Fanuc KAREL source: ko00023.KL

-- PROVISIONAL review KL for V1013-1; original PC SHA256 bdae2d59f309a1ab0a29936beee89b0a31427c261c2ddde664e6fcefbd9250d4
-- Incomplete behavior may be omitted. Consult companion uncertainty JSON. Do not deploy.
PROGRAM KO00023
%NOLOCKGROUP
-- UNRESOLVED_DECL P1 type=000106
-- UNRESOLVED_DECL P2 type=000106
-- UNRESOLVED_DECL P3 type=000106
-- UNRESOLVED_DECL P4 type=000106
-- UNRESOLVED_DECL OUT type=000106
BEGIN
  -- UNRESOLVED_PC offsets 5-80; opcodes 27,27,49,7E,AD,27,49,7E,AD,27,49,7E,AD,27,49,7E,AD,76,7E,4A
  -- UNRESOLVED_PC offsets 85-89; opcodes 7F
END KO00023
